TYPE (* A Structure with 16 BYTES *)
  (* Version 1.0, 2024-02-21, Franz Höpfinger, HR Agrartechnik GmbH *)
  PACKAGE logiBUS::utils::conversion::types;
  ST64B : STRUCT
    B_00 : BYTE; (* BYTE 00 *)
    B_01 : BYTE; (* BYTE 01 *)
    B_02 : BYTE; (* BYTE 02 *)
    B_03 : BYTE; (* BYTE 03 *)
    B_04 : BYTE; (* BYTE 04 *)
    B_05 : BYTE; (* BYTE 05 *)
    B_06 : BYTE; (* BYTE 06 *)
    B_07 : BYTE; (* BYTE 07 *)
    B_08 : BYTE; (* BYTE 08 *)
    B_09 : BYTE; (* BYTE 09 *)
    B_10 : BYTE; (* BYTE 10 *)
    B_11 : BYTE; (* BYTE 11 *)
    B_12 : BYTE; (* BYTE 12 *)
    B_13 : BYTE; (* BYTE 13 *)
    B_14 : BYTE; (* BYTE 14 *)
    B_15 : BYTE; (* BYTE 15 *)
    B_16 : BYTE; (* BYTE 16 *)
    B_17 : BYTE; (* BYTE 17 *)
    B_18 : BYTE; (* BYTE 18 *)
    B_19 : BYTE; (* BYTE 19 *)
    B_20 : BYTE; (* BYTE 20 *)
    B_21 : BYTE; (* BYTE 21 *)
    B_22 : BYTE; (* BYTE 22 *)
    B_23 : BYTE; (* BYTE 23 *)
    B_24 : BYTE; (* BYTE 24 *)
    B_25 : BYTE; (* BYTE 25 *)
    B_26 : BYTE; (* BYTE 26 *)
    B_27 : BYTE; (* BYTE 27 *)
    B_28 : BYTE; (* BYTE 28 *)
    B_29 : BYTE; (* BYTE 29 *)
    B_30 : BYTE; (* BYTE 30 *)
    B_31 : BYTE; (* BYTE 31 *)
    B_32 : BYTE; (* BYTE 32 *)
    B_33 : BYTE; (* BYTE 33 *)
    B_34 : BYTE; (* BYTE 34 *)
    B_35 : BYTE; (* BYTE 35 *)
    B_36 : BYTE; (* BYTE 36 *)
    B_37 : BYTE; (* BYTE 37 *)
    B_38 : BYTE; (* BYTE 38 *)
    B_39 : BYTE; (* BYTE 39 *)
    B_40 : BYTE; (* BYTE 40 *)
    B_41 : BYTE; (* BYTE 41 *)
    B_42 : BYTE; (* BYTE 42 *)
    B_43 : BYTE; (* BYTE 43 *)
    B_44 : BYTE; (* BYTE 44 *)
    B_45 : BYTE; (* BYTE 45 *)
    B_46 : BYTE; (* BYTE 46 *)
    B_47 : BYTE; (* BYTE 47 *)
    B_48 : BYTE; (* BYTE 48 *)
    B_49 : BYTE; (* BYTE 49 *)
    B_50 : BYTE; (* BYTE 50 *)
    B_51 : BYTE; (* BYTE 51 *)
    B_52 : BYTE; (* BYTE 52 *)
    B_53 : BYTE; (* BYTE 53 *)
    B_54 : BYTE; (* BYTE 54 *)
    B_55 : BYTE; (* BYTE 55 *)
    B_56 : BYTE; (* BYTE 56 *)
    B_57 : BYTE; (* BYTE 57 *)
    B_58 : BYTE; (* BYTE 58 *)
    B_59 : BYTE; (* BYTE 59 *)
    B_60 : BYTE; (* BYTE 60 *)
    B_61 : BYTE; (* BYTE 61 *)
    B_62 : BYTE; (* BYTE 62 *)
    B_63 : BYTE; (* BYTE 63 *)
  END_STRUCT;
END_TYPE
